PROGRAM MAIN
VAR
	tonFlash : TON;
	tDelay	: TIME := T#500MS;
END_VAR

//Opening other POUs
Encoder();
Safety();
Laser();
MC();

//LED Flash control
tonFlash(IN:=NOT tonFlash.Q, PT:=tDelay, Q=>);

END_PROGRAM

(* stored: Version 1.1.0.1, ProductVersion 3.1.4024.11
   POU MAIN: Id {d38ddc88-20e8-4c06-9049-cd007a78ceeb}, SpecialFunc None *)
